FUNCTION_BLOCK Preparador_Polimero (* Composite Function Block Type *)
  (* Standard: 61499-2 *)
  (* Version 0.0, 30/03/2026, template *)
  PACKAGE Hidryco.HidrycoLib;
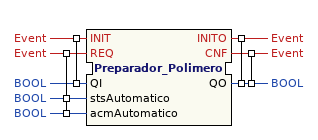
  EVENT_INPUT
    INIT WITH QI; (* Initialization Request *)
    REQ WITH acmAutomatico, stsAutomatico; (* Normal Execution Request *)
  END_EVENT
  EVENT_OUTPUT
    INITO WITH QO; (* Initialization Confirm *)
    CNF WITH QO; (* Execution Confirmation *)
  END_EVENT
  VAR_INPUT
    QI : BOOL; (* Input event qualifier *)
    stsAutomatico : BOOL;
    acmAutomatico : BOOL;
  END_VAR
  VAR_OUTPUT
    QO : BOOL; (* Output event qualifier *)
  END_VAR
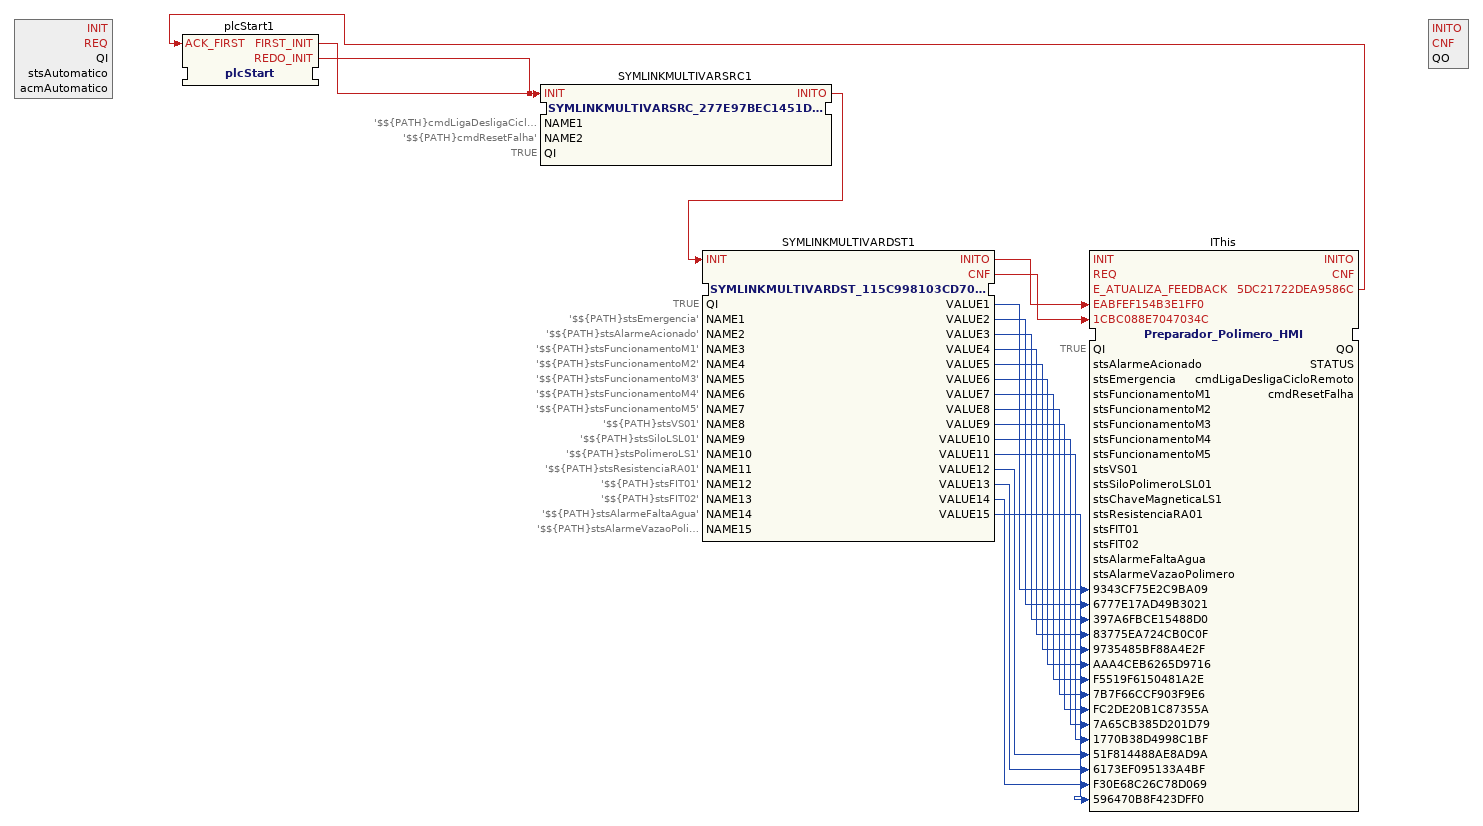
  FBS
    IThis : Preparador_Polimero_HMI(QI := TRUE);
    SYMLINKMULTIVARSRC1 : SYMLINKMULTIVARSRC_277E97BEC1451D2C(NAME1 := '$${PATH}cmdLigaDesligaCicloRemoto', NAME2 := '$${PATH}cmdResetFalha', QI := TRUE); {SET_ATTRIBUTE(Configuration.GenericFBType.InterfaceParams, Runtime.System#I:=2;VALUE${I$}:BOOL,BOOL)}
    SYMLINKMULTIVARDST1 : SYMLINKMULTIVARDST_115C998103CD7017B(QI := TRUE, NAME1 := '$${PATH}stsEmergencia', NAME2 := '$${PATH}stsAlarmeAcionado', NAME3 := '$${PATH}stsFuncionamentoM1', NAME4 := '$${PATH}stsFuncionamentoM2', NAME5 := '$${PATH}stsFuncionamentoM3', NAME6 := '$${PATH}stsFuncionamentoM4', NAME7 := '$${PATH}stsFuncionamentoM5', NAME8 := '$${PATH}stsVS01', NAME9 := '$${PATH}stsSiloLSL01', NAME10 := '$${PATH}stsPolimeroLS1', NAME11 := '$${PATH}stsResistenciaRA01', NAME12 := '$${PATH}stsFIT01', NAME13 := '$${PATH}stsFIT02', NAME14 := '$${PATH}stsAlarmeFaltaAgua', NAME15 := '$${PATH}stsAlarmeVazaoPolimero'); {SET_ATTRIBUTE(Configuration.GenericFBType.InterfaceParams, Runtime.System#I:=15;VALUE${I$}:INT,INT,INT,INT,INT,INT,INT,INT,INT,INT,INT,INT,INT,INT,INT)}
    plcStart1 : plcStart;
  END_FBS
  EVENT_CONNECTIONS
    SYMLINKMULTIVARSRC1.INITO TO SYMLINKMULTIVARDST1.INIT;
    plcStart1.FIRST_INIT TO SYMLINKMULTIVARSRC1.INIT;
    plcStart1.REDO_INIT TO SYMLINKMULTIVARSRC1.INIT;
    SYMLINKMULTIVARDST1.INITO TO IThis.EABFEF154B3E1FF0;
    SYMLINKMULTIVARDST1.CNF TO IThis.1CBC088E7047034C;
    IThis.5DC21722DEA9586C TO plcStart1.ACK_FIRST;
  END_CONNECTIONS
  DATA_CONNECTIONS
    SYMLINKMULTIVARDST1.VALUE1 TO IThis.9343CF75E2C9BA09;
    SYMLINKMULTIVARDST1.VALUE2 TO IThis.6777E17AD49B3021;
    SYMLINKMULTIVARDST1.VALUE3 TO IThis.397A6FBCE15488D0;
    SYMLINKMULTIVARDST1.VALUE4 TO IThis.83775EA724CB0C0F;
    SYMLINKMULTIVARDST1.VALUE5 TO IThis.9735485BF88A4E2F;
    SYMLINKMULTIVARDST1.VALUE6 TO IThis.AAA4CEB6265D9716;
    SYMLINKMULTIVARDST1.VALUE7 TO IThis.F5519F6150481A2E;
    SYMLINKMULTIVARDST1.VALUE8 TO IThis.7B7F66CCF903F9E6;
    SYMLINKMULTIVARDST1.VALUE9 TO IThis.FC2DE20B1C87355A;
    SYMLINKMULTIVARDST1.VALUE10 TO IThis.7A65CB385D201D79;
    SYMLINKMULTIVARDST1.VALUE11 TO IThis.1770B38D4998C1BF;
    SYMLINKMULTIVARDST1.VALUE12 TO IThis.51F814488AE8AD9A;
    SYMLINKMULTIVARDST1.VALUE13 TO IThis.6173EF095133A4BF;
    SYMLINKMULTIVARDST1.VALUE14 TO IThis.F30E68C26C78D069;
    SYMLINKMULTIVARDST1.VALUE15 TO IThis.596470B8F423DFF0;
  END_CONNECTIONS
END_FUNCTION_BLOCK
